FUNCTION_BLOCK FeedOC (* CAT Function Block Type *)
  (* Standard: 61499-2 *)
  (* Version 0.0, 6/7/2026, Schneider Electric, template *)
  PACKAGE SE.Nereda;
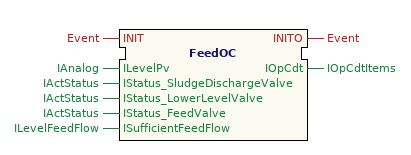
  EVENT_INPUT
    INIT;
  END_EVENT
  EVENT_OUTPUT
    INITO;
  END_EVENT
  SOCKETS
    ILevelPv : IAnalog;
    IStatus_SludgeDischargeValve : IActStatus;
    IStatus_LowerLevelValve : IActStatus;
    IStatus_FeedValve : IActStatus;
    ISufficientFeedFlow : ILevelFeedFlow;
  END_SOCKETS
  PLUGS
    IOpCdt : IOpCdtItems;
  END_PLUGS
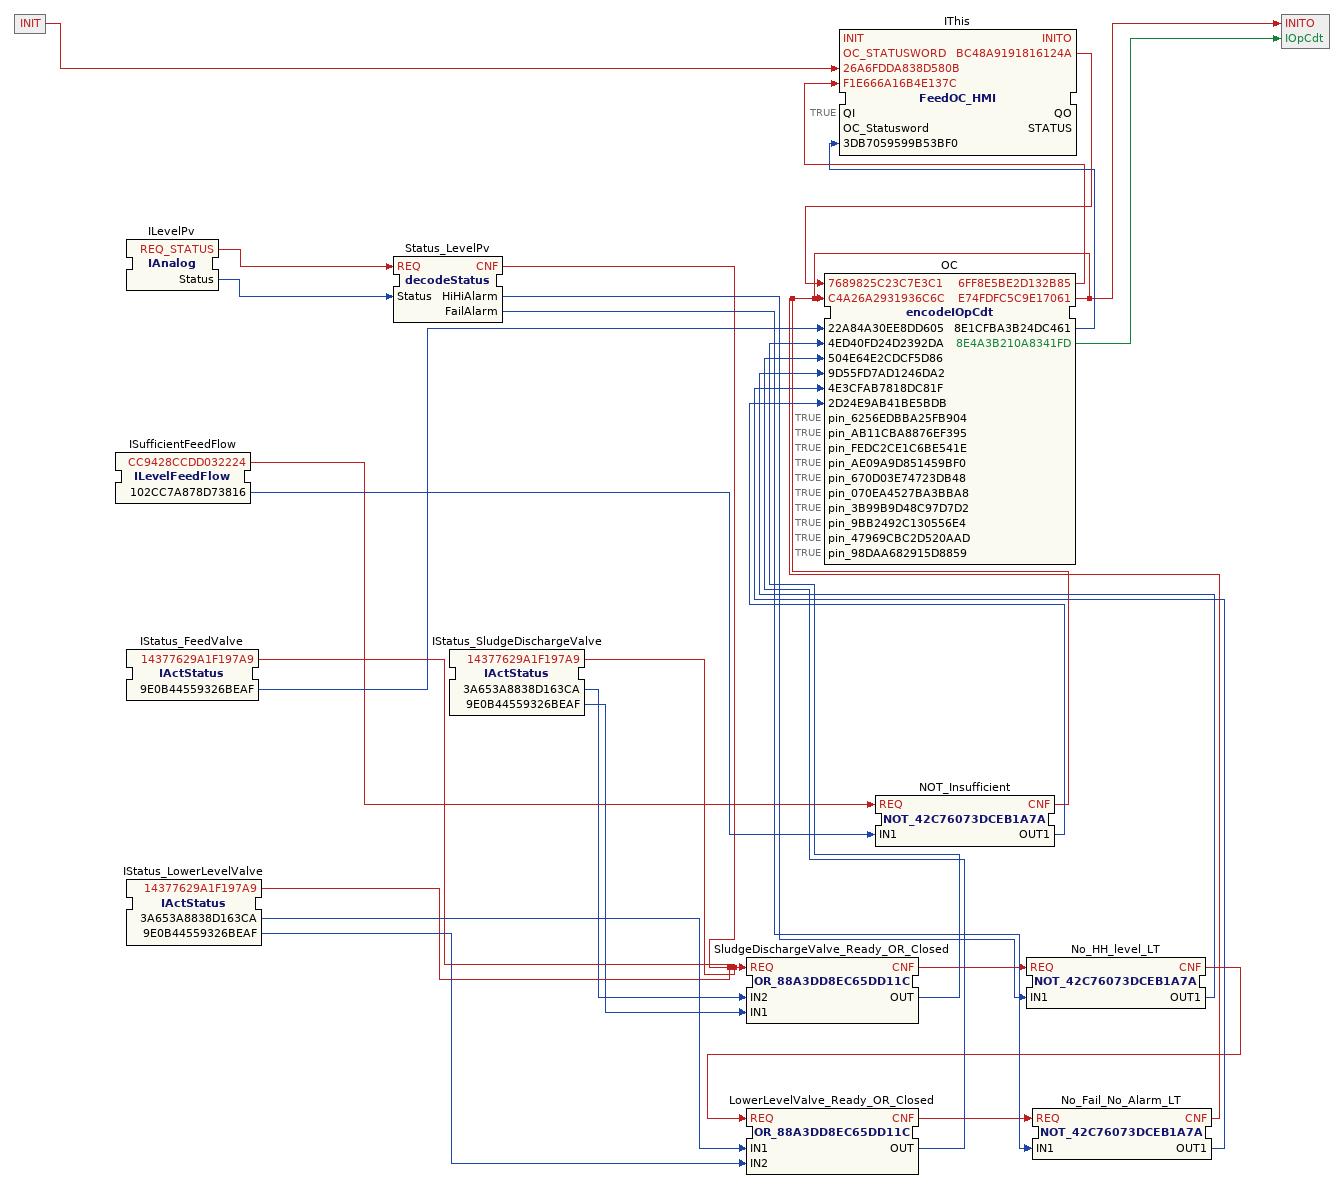
  (* 01 - FUNCTIONNAL INPUT INTERFACE *)
  (* 00 - INITIALIZATION *)
  (* 05 - LOGIC *)
  (* 06 - HMI INTERFACE *)
  (* 03 - FIELD INTERFACE *)
  (* 02 - FUNCTIONNAL OUTPUT INTERFACE *)
  (* Operating Condition Status *)
  (* Operating conditions : 1. Feed valve AV41101 is available 2. Sludge discharge valve AV41103 is available OR closed 3. Lower level valve AV41102 is available OR closed 5. No HH-level (feed) in the reactor 41LT1005 6. Level measurement 41LT1005 available 7. Reserved, do not use 8. Sufficient feed flow *)
  (* Actuators Tags : - Feed valve :                                  AV4x101 - Lower level valve :                        AV4x102 - Air fill valve sludge discharge :    AV4x171 - Chemicals valve :                         AV4x108 - Discharge valve :                         AV4x103 - Vent aeration grid valve :             AV4x107 - Vent sludge grid valve :               AV4x172 *)
  FBS
    OC : encodeIOpCdt(pin_6256EDBBA25FB904 := TRUE, pin_AB11CBA8876EF395 := TRUE, pin_FEDC2CE1C6BE541E := TRUE, pin_AE09A9D851459BF0 := TRUE, pin_670D03E74723DB48 := TRUE, pin_070EA4527BA3BBA8 := TRUE, pin_3B99B9D48C97D7D2 := TRUE, pin_9BB2492C130556E4 := TRUE, pin_47969CBC2D520AAD := TRUE, pin_98DAA682915D8859 := TRUE); (* You set the operating conditions. For the inputs that are not used set a constant to TRUE. *)
    IThis : FeedOC_HMI(QI := TRUE);
    Status_LevelPv : decodeStatus; {SET_ATTRIBUTE(Configuration.Component.HideUnusedPorts, )}
    SludgeDischargeValve_Ready_OR_Closed : OR_88A3DD8EC65DD11C; {SET_ATTRIBUTE(Configuration.GenericFBType.InterfaceParams, Runtime.Standard#CNT:=2;OUT:BOOL)}
    No_HH_level_LT : NOT_42C76073DCEB1A7A; {SET_ATTRIBUTE(Configuration.GenericFBType.InterfaceParams, Runtime.Standard#CNT:=1;OUT${CNT$}:BOOL)}
    No_Fail_No_Alarm_LT : NOT_42C76073DCEB1A7A; {SET_ATTRIBUTE(Configuration.GenericFBType.InterfaceParams, Runtime.Standard#CNT:=1;OUT${CNT$}:BOOL)}
    LowerLevelValve_Ready_OR_Closed : OR_88A3DD8EC65DD11C; {SET_ATTRIBUTE(Configuration.GenericFBType.InterfaceParams, Runtime.Standard#CNT:=2;OUT:BOOL)}
    NOT_Insufficient : NOT_42C76073DCEB1A7A; {SET_ATTRIBUTE(Configuration.GenericFBType.InterfaceParams, Runtime.Standard#CNT:=1;OUT${CNT$}:BOOL)}
  END_FBS
  EVENT_CONNECTIONS
    INIT TO IThis.26A6FDDA838D580B;
    ILevelPv.REQ_STATUS TO Status_LevelPv.REQ;
    Status_LevelPv.CNF TO SludgeDischargeValve_Ready_OR_Closed.REQ;
    SludgeDischargeValve_Ready_OR_Closed.CNF TO No_HH_level_LT.REQ;
    No_HH_level_LT.CNF TO LowerLevelValve_Ready_OR_Closed.REQ;
    OC.6FF8E5BE2D132B85 TO IThis.F1E666A16B4E137C;
    IThis.BC48A9191816124A TO OC.7689825C23C7E3C1;
    IStatus_FeedValve.14377629A1F197A9 TO SludgeDischargeValve_Ready_OR_Closed.REQ;
    IStatus_SludgeDischargeValve.14377629A1F197A9 TO SludgeDischargeValve_Ready_OR_Closed.REQ;
    IStatus_LowerLevelValve.14377629A1F197A9 TO SludgeDischargeValve_Ready_OR_Closed.REQ;
    No_Fail_No_Alarm_LT.CNF TO OC.C4A26A2931936C6C;
    OC.E74FDFC5C9E17061 TO OC.C4A26A2931936C6C;
    OC.E74FDFC5C9E17061 TO INITO;
    LowerLevelValve_Ready_OR_Closed.CNF TO No_Fail_No_Alarm_LT.REQ;
    ISufficientFeedFlow.CC9428CCDD032224 TO NOT_Insufficient.REQ;
    NOT_Insufficient.CNF TO OC.C4A26A2931936C6C;
  END_CONNECTIONS
  DATA_CONNECTIONS
    ILevelPv.Status TO Status_LevelPv.Status;
    Status_LevelPv.HiHiAlarm TO No_HH_level_LT.IN1;
    Status_LevelPv.FailAlarm TO No_Fail_No_Alarm_LT.IN1;
    OC.8E1CFBA3B24DC461 TO IThis.3DB7059599B53BF0;
    IStatus_SludgeDischargeValve.3A653A8838D163CA TO SludgeDischargeValve_Ready_OR_Closed.IN2;
    IStatus_SludgeDischargeValve.9E0B44559326BEAF TO SludgeDischargeValve_Ready_OR_Closed.IN1;
    IStatus_FeedValve.9E0B44559326BEAF TO OC.22A84A30EE8DD605;
    SludgeDischargeValve_Ready_OR_Closed.OUT TO OC.4ED40FD24D2392DA;
    IStatus_LowerLevelValve.3A653A8838D163CA TO LowerLevelValve_Ready_OR_Closed.IN1;
    IStatus_LowerLevelValve.9E0B44559326BEAF TO LowerLevelValve_Ready_OR_Closed.IN2;
    LowerLevelValve_Ready_OR_Closed.OUT TO OC.504E64E2CDCF5D86;
    No_HH_level_LT.OUT1 TO OC.9D55FD7AD1246DA2;
    No_Fail_No_Alarm_LT.OUT1 TO OC.4E3CFAB7818DC81F;
    ISufficientFeedFlow.102CC7A878D73816 TO NOT_Insufficient.IN1;
    NOT_Insufficient.OUT1 TO OC.2D24E9AB41BE5BDB;
  END_CONNECTIONS
  ADAPTER_CONNECTIONS
    OC.8E4A3B210A8341FD TO IOpCdt;
  END_CONNECTIONS
END_FUNCTION_BLOCK
